(* CODESYS project EAS_ELEMENTS.library
   Company: ESCARRE AUTOMATIZACION Y SERVICIOS sl
   Description: Elementos para configurar estructuras de maquinas.
   Version: 0.0.1
   Placeholder: EAS_ELEMENTS
   Author: EAS
   Title: EAS ELEMENTS

Project tree, tasks and I/O mapping:
  libraries: Tc2_Standard, * (Beckhoff Automation GmbH); Tc2_SUPS, * (Beckhoff Automation GmbH); Tc2_System, * (Beckhoff Automation GmbH); Tc2_Utilities, * (Beckhoff Automation GmbH); Tc3_Module, * (Beckhoff Automation GmbH); Util, * (System)
  DUTs/
    DUT Elements/
      data type dutAIn
      data type dutAOut
      data type dutPul
      data type dutPump
      data type dutValve
  GVLs/
  POUs/
    FB Duts/
      function block fAI [ST]
      function block fAO [ST]
      function block fCaudal [ST]
      function block fCnt [ST]
      function block fMotorA [ST]
      function block fOptiDriveP2 [ST]
      function block fPump [ST]
      function block fTemp [ST]
      function block fValve [ST]
*)

// DUTs/DUT Elements/dutAIn
TYPE dutAIn :
STRUCT
iAnalog:INT;	           //Lectura directa analógica

rAna_min: REAL := 0;       //Valor% mínimo analógica 
rAna_max: REAL := 100;	   //Valor% máximo analógica (2V -> 20%)
rUf_min: REAL :=0;		   //Valor mínimo conversión uf
rUf_max: REAL:=100;        //Valor máximo conversión uf

rValue: REAL;			   //Out análogica en UF


END_STRUCT
END_TYPE

// DUTs/DUT Elements/dutAOut
TYPE dutAOut :
STRUCT

// in
rValueUF:REAL;	            //Lectura en UF
rUf_min: REAL := 0;       	//Valor mínimo entrada UF
rUf_max: REAL := 100;  		//Valor máximo entrada UF
rAna_min: REAL :=0;		  	//Valor mínimo conversión Analógica
rAna_max: REAL:=32767;      //Valor máximo conversión Analógica

//out
rAnalog: REAL;			    //Out análogica
iAnalog: INT;			    //Out análogica

END_STRUCT
END_TYPE

// DUTs/DUT Elements/dutPul
TYPE dutPul :
STRUCT
	xPul:BOOL;		// IN Pulsador
	xPil:BOOL;		// OUT Piloto

END_STRUCT
END_TYPE

// DUTs/DUT Elements/dutPump
TYPE dutPump :
STRUCT
	xInRun:BOOL;		//In Forware Pump
	xInRev:BOOL;		//In Reverse Pump
	rSPVelFoward:REAL;	//In Speed reference 
	rSPVelRevers:REAL;	//In Speed reference 
	xInCons:BOOL;		//In OK Pump
	xInFail:BOOL;		//In Fail Pump
	
	xFoward:BOOL;		(*Run Foward*)
	xReverse:BOOL;		(*Run Reverse*)	
	rSpeed:REAL;		(*Vel to inverter*)

	xOK:BOOL;			(*Pump Run OK*)
	xFailOut:BOOL;		(*Fail Pump*)
	xNo_Ok:BOOL;		(*Falta consenso*)
	
END_STRUCT
END_TYPE

// DUTs/DUT Elements/dutValve
TYPE dutValve :
STRUCT
	
xOpen: BOOL;		// Salida activa vávlula
xFCo: BOOL;			// In FC NO
xFCc: BOOL;			// IN FC NC
xFailFCo: BOOL;		// Out fallo FC NO
xFailFCc: BOOL;		// Out fallo FC NC
xFailFC: BOOL;		// Out fallo FC

END_STRUCT
END_TYPE

// POUs/FB Duts/fAI
FUNCTION_BLOCK fAI
VAR_IN_OUT
	Ai:dutAIn;
END_VAR


VAR
	rAna_min: REAL := 0;
	rAna_MAX: REAL := 32767;
	bCre: BOOL;
END_VAR

(*-------------------------------------------------------------------------------------------------------*)

	(*Comprobar lectura creciente o decreciente*)
IF AI.rAna_min < AI.rAna_max THEN
		bCre:=TRUE; 
		ELSE
		bCre:=FALSE;
END_IF


	(*valores min y maximo de la analogica*)
IF bCre 
	THEN
		rAna_min:=(((AI.rAna_min)/100.0)*32767);
		rAna_max:=(((AI.rAna_max)/100.0)*32767);
	ELSE
		rAna_max:=(((AI.rAna_min)/100.0)*32767);
		rAna_min:=(((AI.rAna_max)/100.0)*32767);
END_IF

	(*Buscar valor de lectrua analogico*)
	(*Carregar lectura percentual *)
	AI.rValue:=Canvi_Escala(
			In:= AI.iAnalog, 
			In_Min:= rAna_min, 
			In_Max:= rAna_max, 
			Out_Min:= AI.rUf_min, 
			Out_Max:= AI.rUf_max);

END_FUNCTION_BLOCK

// POUs/FB Duts/fAO
FUNCTION_BLOCK fAO
VAR_IN_OUT
	AO:dutAOut;
END_VAR

VAR
	
END_VAR

(*-------------------------------------------------------------------------------------------------------*)



AO.rAnalog:= Canvi_Escala(
			In:= AO.rValueUF, 
			In_Min:= AO.rUf_min, 
			In_Max:= Ao.rUf_max, 
			Out_Min:= AO.rAna_min, 
			Out_Max:= AO.rAna_max);

AO.iAnalog:= REAL_TO_INT(AO.rAnalog);

END_FUNCTION_BLOCK

// POUs/FB Duts/fCaudal
FUNCTION_BLOCK fCaudal
VAR_INPUT
	///Posicion del contador
	iCnt: UDINT;
	///Reset Contador
	xReset: BOOL;
	///PF Frecuencia maxima caudalimetro Hz
	iPFFrec: INT;
	///PF Caudal a la freq maxima lit/min
	iPFFlowMax: INT;
	///PF Tiempo para el calculo de lcaudal
	iPFTmClcFlow: TIME;
END_VAR
VAR_OUTPUT
	///Acumulado litros
	rLit: REAL;
	///Valor instantaneo Caudal
	rFlow: REAL;
END_VAR
VAR
	iCnt_acu: UDINT;
	iPulsos: UDINT;
	iprueba: UDINT;
	imax: UDINT;
	imanual: UDINT;
	xresetMan: BOOL;
END_VAR


//Reset 
IF xReset OR xresetMan
 THEN
	iCnt_acu:=iCnt;
END_IF
iPulsos :=iCnt-iCnt_acu;

iprueba:= imax - imanual;

//Calculo Litros -----------------------------------------
//asegurar que el divisor tiene valor
IF iPFFrec=0 THEN
	iPFFrec:=1000;
END_IF

rLit:= (UDINT_TO_REAL(iPulsos)*iPFFlowMax)/(iPFFrec*60);



//Calculo Caudal    FALTA

END_FUNCTION_BLOCK

// POUs/FB Duts/fCnt
FUNCTION_BLOCK fCnt
VAR_INPUT
	///Valor contador
	iCnt: UDINT;
END_VAR

(*Entrada tipo 1008 BECHOFF CNT*)

END_FUNCTION_BLOCK

// POUs/FB Duts/fMotorA
FUNCTION_BLOCK fMotorA
VAR_INPUT
	xRun:BOOL;
	xPantallaVestir:bool;
END_VAR
VAR_OUTPUT
END_VAR
VAR_IN_OUT
	MotorA:dutMotorArrastre;

END_VAR

VAR
	t_fc_fail: Ton;
	PercentCopm: REAL;
	ValorAjustMax: REAL;
	rSP_Speed_mt_min: INT;
	RS_FailFC: Rs;
END_VAR

//NUMERO MOTOR DE ARRASTRE


//=============================================
// Poner en marcha
//==============================================
//adelante
MotorA.xFoward:= (MotorA.xPulFoward AND
						 xRun) ;

//Atras
MotorA.xRevers:= MotorA.xPulRevers AND
						xRun;


//============================================
// CAlculo velocidad
//============================================
IF MotorA.iPF_CompInv=0
	THEN
	MotorA.rDiferenciaComp:=MotorA.rCompRef- MotorA.rCompensator.rValue;
	ELSE
	MotorA.rDiferenciaComp:=MotorA.rCompensator.rValue-MotorA.rCompRef;	
END_IF
PercentCopm:=MotorA.rDiferenciaComp/50.0;
ValorAjustMax:=(INT_TO_REAL(MotorA.iPF_FactorCompensador)*MotorA.rSPSpeedMac/100.0);

MotorA.rAjustVel:= PercentCopm*ValorAjustMax;



// Forzar velocidad a cero si se esta en pantalla de vestir
IF xPantallaVestir AND NOT(MotorA.xPulRunMan) 
	THEN
	MotorA.rSpeedMot.rValueUF:=0;
	ELSE
	MotorA.rSpeedMot.rValueUF:= MotorA.rSPSpeedMac+MotorA.rAjustVel;
END_IF
//$$$$$$$$$$$$$$$$$$$$$$$$$$$$$$$$$$$$$$$$$$$$$$$$$$$$$$$$$$$$$$$$$$$$$$$$
//============================================
// FALLO FC
//============================================

MotorA.xFC_OK:= (MotorA.xFC_Down AND MotorA.xFC_Up) OR motorA.xFC_inOK;

t_fc_fail(IN:=NOT(MotorA.xFC_OK) AND xRun , PT:=MotorA.time_FailFC);
RS_FailFC(SET:= t_fc_fail.Q, RESET1:=motorA.xResetFail );


MotorA.xAlarmFC:=RS_FailFC.Q1;

END_FUNCTION_BLOCK

// POUs/FB Duts/fOptiDriveP2
FUNCTION_BLOCK fOptiDriveP2
VAR_INPUT
	xForward:BOOL;		(*PDI Word 1: bit0	Drive Run Foward*)
	xRevers:BOOL;		(*PDI Word 1: bit0 	Drive Run Reverde*)
	xFastStop:BOOL;		(*PDI Word 1: bit1	Drive Stop with Deceleration Ramp 2*)
	xFaultReset:BOOL;	(*PDI Word 1: bit2*	Rising Edge fault reset request*)
	xCoastStop:BOOL;	(*PDI Word 1: bit3	Drive Coasts to stop. Overrides bit 0 *)
	rSetPointFreq:REAL;	(*PDI Word 2: Fixed Function : Frequency Setpoint 500-> 50Hz *)
	rWord3:REAL;		(*PDI Word 3 : User Defined Function  P5-14*)
	rWord4:REAL;		(*PDI Word 4 : User Defined Function  P5-13*)
END_VAR

VAR_OUTPUT
	xRunOK:BOOL;		(*PD0 Word 1: bit0   Indicates when the output to the motor is enabled *)
	XFault:BOOL;		(*PD0 Word 1: bit1   Indicates when the drive has tripped. *)
	xHandMode:BOOL;		(*PD0 Word 1: bit2   Optidrive HVAC Only. Indicates when Hand control is selected  *)
	xInhibit:BOOL;		(*PD0 Word 1: bit3   Indicates the status of the STO / Hardware Inhibit circuit  *)
	xMaintenTime:BOOL;	(*PD0 Word 1: bit4   Indicates that the programmable System Maintenance Time Interval has expired  *)
	bLastFail:INT;		(*PD0 Word 1: bit8-15 Indicates the last or current fault code *)
	rOutFreq:REAL;		(*PDO Word 2: Fixed Function : Output Frequency*)
	rOutCurrent:REAL;	(*PDO Word 3: Default:Output Current. Data to be transferred in this word can be selected by the User in drive parameter P5-12 *)
	rOutWord4:REAL;		(*PDO Word 4 : User Defined. Data to be transferred in this word can be selected by the User in drive parameter P5-08*)
	
END_VAR
VAR_IN_OUT
	Variador:dutOptidriveP2;
END_VAR
VAR

	iAux1: INT;
	iAux2: INT;
	AuxFail1: WORD;
	AuxFail2: word;
END_VAR

// CONTROL: Entradas al variador

//word 1 -----------------------------------------------------------

variador.CONTROL[1]:=DWORD_TO_WORD(putbit(variador.CONTROL[1],0,(xForward OR xRevers)));
variador.CONTROL[1]:=DWORD_TO_WORD(putbit(variador.CONTROL[1],1,xFastStop));
variador.CONTROL[1]:=DWORD_TO_WORD(putbit(variador.CONTROL[1],2,xFaultReset));
variador.CONTROL[1]:=DWORD_TO_WORD(putbit(variador.CONTROL[1],3,xCoastStop));



//Word 2 -----------------------------------------------------------
//Marcha Directa
variador.CONTROL[2]:= 0;
IF xForward
	THEN
	variador.CONTROL[2]:= REAL_TO_WORD(rSetPointFreq*10);
END_IF
//Marcha Inversa
IF xRevers
	THEN
	iAux1:= REAL_TO_INT(rSetPointFreq*10) ;
	iAux2:= iAux1*-1;
	variador.CONTROL[2]:= iAux2;   (*FORZAMOS UN INT EN UN WORD PARA PODER REALIZAR EL NEGATIVO*)
END_IF

//variador.CONTROL[2]:= REAL_TO_WORD(rSetPointFreq*10);


//Word 3 -----------------------------------------------------------
variador.CONTROL[3]:= REAL_TO_WORD(rWord3);

//Word 4 -----------------------------------------------------------
variador.CONTROL[4]:= REAL_TO_WORD(rWord4);



//STATUS: Salidas Variador

//word 1 -----------------------------------------------------------

xRunOK			:=EXTRACT(variador.STATUS[1],0);
XFault			:=EXTRACT(variador.STATUS[1],1);
xHandMode		:=EXTRACT(variador.STATUS[1],2);
xInhibit		:=EXTRACT(variador.STATUS[1],3);
xMaintenTime	:=EXTRACT(variador.STATUS[1],4);


//Last Fail
bLastFail:= WORD_TO_INT(SHR(variador.STATUS[1],8));
	

//Word 2 -----------------------------------------------------------
rOutFreq:= WORD_TO_REAL(variador.STATUS[2])/10.0;

//Word 3 -----------------------------------------------------------
rOutCurrent:= WORD_TO_REAL(variador.STATUS[3]);

//Word 4 -----------------------------------------------------------
rOutWord4:= WORD_TO_REAL(variador.STATUS[4]);

END_FUNCTION_BLOCK

// POUs/FB Duts/fPump
FUNCTION_BLOCK fPump

VAR_IN_OUT
	pump:dutPump;
END_VAR

VAR
	a: INT;
	ton_NoOk: Ton;
END_VAR

a:=a+1;

//marcha adelante
pump.xFoward:= pump.xInRun AND NOT(pump.xInRev) AND NOT(pump.xFailOut);

//marcha Atras
pump.xReverse:= pump.xInRun AND NOT(pump.xInRev)AND NOT(pump.xFailOut);

//velocidad
pump.rSpeed:=0;
IF pump.xFoward THEN
	pump.rSpeed:=pump.rSPVelFoward;
END_IF
IF pump.xReverse THEN
	pump.rSpeed:=pump.rSPVelRevers;
END_IF

//Indicacion Bomba ok (Bomba girando)
pump.xOK:= (pump.xFoward OR pump.xReverse ) AND pump.xInCons  ;

//Alarma Falta consenso
ton_NoOk(IN:=(pump.xFoward OR pump.xReverse ) AND NOT(pump.xInCons) , PT:= T#5S );
pump.xNo_Ok := ton_NoOk.Q  ;

//Alarma Fallo Variador
pump.xFailOut:= pump.xInFail;

END_FUNCTION_BLOCK

// POUs/FB Duts/fTemp
FUNCTION_BLOCK fTemp
VAR_IN_OUT
	Ai:dutAIN;
END_VAR


VAR
END_VAR

(*-------------------------------------------------------------------------------------------------------*)
(*Conversion UF a temperatura ºC*)
Ai.rValue :=INT_TO_REAL(Ai.iAnalog)/10.0;

END_FUNCTION_BLOCK

// POUs/FB Duts/fValve
FUNCTION_BLOCK fValve

VAR_IN_OUT
	valv:dutValve;
END_VAR

VAR
	a: INT;
	tonFailFCOp: Ton;
	tonFailFCCl: Ton;
	bFailFCop:BOOL;	(*Fail FC*)
	bFailFCcl:BOOL;	(*Fail FC*)
	test: BOOL;
	tToFail: TIME := T#5S;
END_VAR

a:=a+1;

valv.xFailFC:=FALSE;
valv.xFailFCc:=FALSE;
valv.xFailFCo:=FALSE;
		
(*=========================================================================================================*)
(*Salida  BECHOFF DO*)
				
(*FC valve open*)
tonFailFCOp(IN:= (valv.xOpen)AND NOT(valv.xFailFCo) , PT:=tToFail );
valv.xFailFCo:= tonFailFCOp.Q;

(*FC valve close*)
tonFailFCCl(IN:= NOT(valv.xOpen)AND NOT(valv.xFailFCc) , PT:=tToFail  );
valv.xFailFCc:= tonFailFCCl.Q;

(*FC Valve*)		
valv.xFailFC:= valv.xFailFCo OR valv.xFailFCc;

(*=========================================================================================================*)

END_FUNCTION_BLOCK
